FUNCTION_BLOCK FB_PersistentDataManager
VAR PERSISTENT
    _PanelFrontLength : REAL;
    _Config           : ST_RecipeBuilder_Config;
    _GantryConfig     : ST_GantryXYZ_Config; 
END_VAR

PROPERTY Config : ST_RecipeBuilder_Config
GET
Config := _Config;
END_GET
SET
_Config := Config;
END_SET
END_PROPERTY

PROPERTY GantryConfig : ST_GantryXYZ_Config
GET
GantryConfig := _GantryConfig;
END_GET
SET
_GantryConfig := GantryConfig;
END_SET
END_PROPERTY

END_FUNCTION_BLOCK

(* stored: Version 1.1.0.1, ProductVersion 3.1.4024.15
   POU FB_PersistentDataManager: Id {4ed47747-e9e7-4807-96fb-1abdb1959994}, SpecialFunc None
   Property Config: Id {1a5d92ef-6b65-43a4-903f-d617f66a22f2}
   Get Get: Id {9300e8ec-af0f-4824-bd13-92b6592fc495}
   Set Set: Id {4e6adcec-48a4-45cf-8715-df36f2a76f6a}
   Property GantryConfig: Id {94b2adc8-df4b-49c8-b6d5-478bf602fa4a}
   Get Get: Id {29f79859-4371-4222-88cc-78612130e959}
   Set Set: Id {8ab71232-b490-4947-8d5e-0094c8f735e8} *)
